TYPE ST_WashPoint EXTENDS ST_3DPoint :
STRUCT
	nRinseChannel : USINT;
END_STRUCT
END_TYPE

(* stored: Version 1.1.0.1, ProductVersion 3.1.4020.6
   DUT ST_WashPoint: Id {91859c74-302f-4bf9-9414-d0b50f79ec71} *)
